{attribute 'GeneratedUsingTerminal: EK1101-0000-0016'}
{attribute addProperty BoxType "EK1101-0000-0016"}
{attribute addProperty Id "IDAT %I*UINT2"}
{attribute addProperty CRC "130667151"}
{attribute addProperty Size "2"}
TYPE ID_07C9D28F :
STRUCT
	{attribute addProperty Name "ID"}
	ID AT %I* : UINT;
END_STRUCT
END_TYPE

(* stored: Version 1.2.0.0, ProductVersion 3.1.4024.9
   DUT ID_07C9D28F: Id {54aedcfd-5835-48f0-9c1e-00c7ffed1c9e} *)
